// SIMATIC STEP 7 (V5.x) project EMPTYING
// program: S7 Program(1)

SYMBOL_TABLE
"EMPTYING_CYCLE"	FB 148	FB 148	// Цикл опустошения илоуплотнителей
END_SYMBOL_TABLE

FUNCTION_BLOCK "EMPTYING_CYCLE"	// FB 148
TITLE = Блок управления циклами слива
//Используемая переферия:
//Таймеры:
//Счетчики:
//
//
////Авария по сливу, насосы откачки не запустились
////Фильтр аварий в режимах работы чтобы запустить слив на одном затворе
AUTHOR : ETSystem
VERSION : 0.1
VAR_INPUT
  G32_OPENED : BOOL ;	//Затвор 3-2 открыт
  G32_CLOSED : BOOL ;	//Затвор 3-2 закрыт
  G32_FAULT : BOOL ;	//Авария затвора 3-2
  G34_OPENED : BOOL ;	//Затвор 3-4 открыт
  G34_CLOSED : BOOL ;	//Затвор 3-4 закрыт
  G34_FAULT : BOOL ;	//Авария затвора 3-4
  WT_ONOFF : BOOL ;	//Цикл ожидания активен/нет
  AUTO_ONOFF : BOOL ;	//Автоматический режим включен
  LEVEL_1 : BOOL ;	//Датчик уровня 1 (минимальный уровень)
  LEVEL_2 : BOOL ;	//Датчик уровня 2 (средний уровень)
  LEVEL_3 : BOOL ;	//Датчик уровня 3 (высокий уровень)
  LEVEL_4 : BOOL ;	//Датчик уровня 4 (критический уровень)
  STOP : BOOL ;	//Цикл остановлен
  START : BOOL ;	//Цикл запущен
  EMPTYING_DELAY : INT  := 10;	//Задержка начала слива (в формате TIME)
  G32_CNT_TASK : INT  := 1;	//Количество циклов опорожения затвора 3-2 (0 - 4)
  G34_CNT_TASK : INT  := 1;	//Количество циклов опорожения затвора 3-4 (0 - 4)
END_VAR
VAR_OUTPUT
  QG32_OPENING : BOOL ;	//Команда на открытие затвора 3-2
  QG32_CLOSING : BOOL ;	//Команда на закрытие затвора 3-2
  QG32_FAULT : BOOL ;	//Авария на затворе 3-2
  QG34_OPENING : BOOL ;	//Команда на открытие затвора 3-4
  QG34_CLOSING : BOOL ;	//Команда на закрытие затвора 3-4
  QG34_FAULT : BOOL ;	//Авария на затворе 3-4
  QCOMMON_FAULT : BOOL ;	//Общая авария на блоке
  QINIT_OK : BOOL ;	//Работа цикла слива в автоматическом режиме инициализирована
  QG32_ACK : BOOL ;	//Идет слив с затвора 3-2
  QG34_ACK : BOOL ;	//Идет слив с затвора 3-4
  QEMPTYING_ACK : BOOL ;	//Режим слива активен
  QWORK_TIME : INT ;	//Общее время работы слива
END_VAR
VAR_IN_OUT
  G32_CNT : INT ;	//Счетчик циклов слива (затвор 3-2)
  G34_CNT : INT ;	//Счетчик циклов слива (затвор 3-4)
END_VAR
VAR
  LEVEL_FAULT : BOOL ;	//Неисправность датчика уровня
  GATE_FAULT : BOOL ;	//Неисправность одного из затворов (3-2 или 3-4)
  COMMON_FAULT : BOOL ;	//Общая ошибка
  DELAY_OK : BOOL ;	//Задержка цикла слива отработана
  G32_INWORK : BOOL ;	//Затвор 3-2 в работе
  G34_INWORK : BOOL ;	//Затвор 3-4 в работе
  G32_CNT_FLAG : BOOL ;	//Флаг для подсчета циклов слива (затвор 3-2)
  G34_CNT_FLAG : BOOL ;	//Флаг для подсчета циклов слива (затвор 3-4)
  BOTH_FLAG : BOOL ;	//Оба затвора в работе
  INIT_OK : BOOL ;	//Режим слива инициализирован
  MODE : INT ;	//0 - оба неактивны, 1 - оба активны, 2 - активен 3-2, 3 - активен 3-4
  S5T_EMPDELAY : S5TIME ;	//Задержка начала слива (в формате S5T)
  T_EMPDELAY : TIME ;	//Задержка начала слива (в формате TIME)
END_VAR
BEGIN
NETWORK
TITLE = Инициализация цикла (начало)
//Инициализация цикла необходима только один раз при запуске автоматического 
//режима, если инициализация проходит без ошибок, выставляется флаг INIT_OK и на 
//следующем цикле ПЛК готов к автоматическому сливу из илоуплотнителей
//Мы не в автоматическом режиме, уходим сбросив инициализацию цикла если он была
      AN    #AUTO_ONOFF;
//Сбросим признаки аварии после того как выбило в ручной режим
      R     #COMMON_FAULT;
      R     #QCOMMON_FAULT;
      JC    MAN;
//Сбросим сигналы открытия/закрытия если требуется: 
//Сброс сигналов открытия/закрытия  32
      A     #QG32_OPENING;
      A     #G32_OPENED;
      O(;
      A     #QG32_OPENING;
      AN    #G32_OPENED;
      AN    #G32_CLOSED;
      );
      R     #QG32_OPENING;
      A     #QG32_CLOSING;
      A     #G32_CLOSED;
      O(;
      A     #QG32_CLOSING;
      AN    #G32_OPENED;
      AN    #G32_CLOSED;
      );
      R     #QG32_CLOSING;
//Сброс сигналов открытия/закрытия 34
      A     #QG34_OPENING;
      A     #G34_OPENED;
      O(;
      A     #QG34_OPENING;
      AN    #G34_OPENED;
      AN    #G34_CLOSED;
      );
      R     #QG34_OPENING;
      A     #QG34_CLOSING;
      A     #G34_CLOSED;
      O(;
      A     #QG34_CLOSING;
      AN    #G34_OPENED;
      AN    #G34_CLOSED;
      );
      R     #QG34_CLOSING;
//Определяем состояние автоматического режима
      A     #START;
      AN    #INIT_OK;
      JC    INIT;
      AN    #START;
      JC    STOP;
      A     #INIT_OK;
      JC    AUTO;
      JU    N1;
NETWORK
TITLE =  Инициализация цикла (продолжение)
//Выбор верной конфигурации затворов слива:
//Определяем конфигурацию системы слива (единожды). Возможные варианты:
// 1. Активны оба затвора (G32_CNT и G34_CNT) - число их циклов слива не равно 0 
//(MODE 0), выставляется флаг BOTH_FLAG.
// 2. Активен один из затворов (G32_CNT ИЛИ G34_CNT) - число его циклов слива 
//равно 0 (MODE 1, MODE 2).
// 3. Слив запрещен (MODE 0).
// 4. Запись значения в MODE выводится для более удобного наблюдения за тем какой 
//режим был проинициализирован. (для отладки) 
//
//Смена конфигурации режима работы сливов во время исполнения автоматического 
//режима не предусмотрена, и будет инициализирована авария. (Так же она должна 
//быть заблокирована в СКАДА).
//Инициализация (сброс) флагов
INIT: NOP   0;
      L     0;
      T     #G32_CNT;
      T     #G34_CNT;
      SET;
      R     #G32_CNT_FLAG;
      R     #G34_CNT_FLAG;
      R     #G32_INWORK;
      R     #G34_INWORK;
//Сбросим признаки аварии при инициализации
      R     #COMMON_FAULT;
      R     #QCOMMON_FAULT;
//Закроем затворы если открыты:
      AN    #G32_CLOSED;
      S     #QG32_CLOSING;
      AN    #G34_CLOSED;
      S     #QG34_CLOSING;
//Оба затвора могут быть в работе (MODE 1)
      AN    #G32_FAULT;
      AN    #G34_FAULT;
      A(;
      L     #G32_CNT_TASK;
      L     0;
      <>I;
      );
      A(;
      L     #G34_CNT_TASK;
      L     0;
      <>I;
      );
      L     1;
//Инициализаруем активный затвор и флаг того что
//в работе оба затвора
      S     #G32_INWORK;
      S     #BOTH_FLAG;
      JC    MSEL;
//Затвор 3-2 может быть в работе (MODE 2)
      AN    #G32_FAULT;
      A(;
      L     #G32_CNT_TASK;
      L     0;
      <>I;
      );
      L     2;
      S     #G32_INWORK;
      R     #BOTH_FLAG;
      JC    MSEL;
//Затвор 3-4 может быть в работе (MODE 3)
      AN    #G34_FAULT;
      A(;
      L     #G34_CNT_TASK;
      L     0;
      <>I;
      );
      L     3;
      S     #G34_INWORK;
      R     #BOTH_FLAG;
      JC    MSEL;
//Ни один из затворов в работе быть не может (MODE 0)
      L     0;
//Задание активной конфигурации
MSEL: T     #MODE;
//Если режим MODE = 0, пропускаем цикл опустошения:
      L     #MODE;
      L     0;
      ==I;
      JC    MOD0;
NETWORK
TITLE =  Инициализация цикла (продолжение)
//Конвертация времени ожидания перед сливом из INT (SCADA) в S5T (Siemens) с 
//помощью функции FC40, через переменную типа TIME (IEC). Итого вое время в 
//секундах. Задание из SCADA в секундах.
      L     #EMPTYING_DELAY;
      ITD;
      L     L#1000;
      *D;
      T     #T_EMPDELAY;
      CALL  FC 40 (
           $1                       := #T_EMPDELAY,
           $2                       := #S5T_EMPDELAY);
NETWORK
TITLE = Инициализация цикла слива (конец)
//Если включен автоматический режим, и бак пуст (не один из датчиков не включен)
      A     #AUTO_ONOFF;
      A     #G32_CLOSED;
      A     #G34_CLOSED;
      AN    #LEVEL_1;
      AN    #LEVEL_2;
      AN    #LEVEL_3;
      AN    #LEVEL_4;
      S     #INIT_OK;
      JCN   N1;
NETWORK
TITLE = Автоматический режим слива илоуплотнителей (начало)
//Сброс сигналов на открытие или закрытие затворов
AUTO: NOP   0;
NETWORK
TITLE = Переинициализация автомата
//Если мы не в режиме ожидания, сбросим таймер и флаг окончания задержки, а так 
//же обнулим счетчики сливов по каждому из затворов.
      AN    #WT_ONOFF;
      R     T 5;
      R     #DELAY_OK;
      JCN   NX1;
//Обнуление счетчиков
      L     0;
      T     #G32_CNT;
      T     #G34_CNT;
//Сброс флагов
      SET;
      R     #G32_CNT_FLAG;
      R     #G34_CNT_FLAG;
//Переинициализация активного затвора
      A     #BOTH_FLAG;
      O(;
      L     #MODE;
      L     2;
      ==I;
      );
      S     #G32_INWORK;
      L     #MODE;
      L     3;
      ==I;
      S     #G34_INWORK;
NETWORK
TITLE = Определение аварий
//Определяем текущие аварии, при их возникновении цикл налива-слива должен быть 
//остановлен, для этого необходимо использовать блок налива (FB_xxx) как блок 
//общей задачи автоматического режима. Вопрос с ручным - автоматическим режимом 
//на затворах 3-2 и 3-4 требует отдельного рассмотрения. 
//
//Подумать над общей неисправностью.
NX1:  NOP   0;
//Проверяем верно ли работает линейка датчиков 
//Неисправность датчика первого уровня:
//(НЕ Уровень1 И (Уровень2 ИЛИ Уровень3 ИЛИ Уровень4))
      AN    #LEVEL_1;
      A(;
      O     #LEVEL_2;
      O     #LEVEL_3;
      O     #LEVEL_4;
      );
      O;
//Или их непоследовательное включение:
//(Уровень1 И ((Уровень3 И НЕ Уровень2) ИЛИ (Уровень4 И НЕ Уровень3))
      A     #LEVEL_1;
      A(;
      A     #LEVEL_3;
      AN    #LEVEL_2;
      O;
      A     #LEVEL_4;
      AN    #LEVEL_3;
      );
      =     #LEVEL_FAULT;
//Проверяем наличие аварий на затворах 3-2 и 3-4:
//Неисправности затворов:
//     O     #G32_FAULT
//      O     #G34_FAULT
//      =     #GATE_FAULT
//Выдаем аварии по затвору в зависимости от режима работы:
//Режим 1:
      L     #MODE;
      L     1;
      ==I;
      JC    ERR1;
//Режим 2:
      L     #MODE;
      L     2;
      ==I;
      JC    ERR2;
//Режим 3:
      L     #MODE;
      L     3;
      ==I;
      JC    ERR3;
//Нет аварий по затворам
      JU    ERRC;
ERR1: NOP   0;
      O     #G32_FAULT;
      O     #G34_FAULT;
      =     #GATE_FAULT;
      JU    ERRC;
ERR2: NOP   0;
      A     #G32_FAULT;
      =     #GATE_FAULT;
      JU    ERRC;
ERR3: NOP   0;
      A     #G34_FAULT;
      =     #GATE_FAULT;
ERRC: NOP   0;
//Общая неисправность:
      O     #LEVEL_FAULT;
      O     #GATE_FAULT;
      =     #COMMON_FAULT;
      JC    ALRM;
NETWORK
TITLE = Задержка начала первого цикла слива
//Если активировался режим ожидания налива (WT_ONOFF = 1) И с определенной 
//конфигурацией (MODE != 0) -  дополнительная проверка, которую можно убрать.
//То запускаем таймер задержки слива (T5 - 
//DELAY_EMPTYING), S_ODT - считает пока на его входе 1, если она пропадает, счет 
//останавливается и при восcтановлении сигнала запускается заново. 
      A     #DELAY_OK;
      JC    NX2;
      A     #WT_ONOFF;
      A(;
      L     #MODE;
      L     0;
      <>I;
      );
      L     #S5T_EMPDELAY;
      SD    T 5;
      A     T 5;
      S     #DELAY_OK;
      S     #QEMPTYING_ACK;
NETWORK
TITLE = Цикл слива с обоих затворов
//В зависимости от режима работы возможно нескольк сценариев слива:
// 1. Через оба клапана, сначала n циклов с 3-2, затем n циклов с 3-4
// 2. n циклов через один клапан (3-2 или 3-4) 
NX2:  NOP   0;
//Если задержка после заполнения не отработала, то начинать процесс слива
//нельзя, ожидаем поднятие флага DELAY_OK
      AN    #DELAY_OK;
      JC    N1;
//Если G32 в работе, инициализируем слив
      A     #G32_INWORK;
      AN    #G32_CNT_FLAG;
      JC    G32E;
//Цикл отработал и затвор закрылся
      A     #G32_CNT_FLAG;
      A     #G32_CLOSED;
      JC    G32C;
//Если G34 в работе, инициализируем слив
      A     #G34_INWORK;
      AN    #G34_CNT_FLAG;
      JC    G34E;
//Цикл отработал и затвор закрылся
      A     #G34_CNT_FLAG;
      A     #G34_CLOSED;
      JC    G34C;
      JU    N1;
//////////////////////Затвор 3-2/////////////////////
//Открытие и закрытие затвора
G32E: NOP   0;
//Открываем затвор если уровень в баке опустился до нужного уровня
//И затвор открыт
      AN    #LEVEL_1;
      A     #G32_CLOSED;
      S     #QG32_OPENING;
      S     #QG32_ACK;
//Закрываем затвор если уровень в баке поднялся до нужного уровня
//И затвор открыт, так же устанавливаем флаг для подсчета циклов
      A     #LEVEL_2;
      A     #G32_OPENED;
      S     #QG32_CLOSING;
      S     #G32_CNT_FLAG;
      JU    N1;
//Подсчет циклов и условие выхода (смены затвора)
G32C: NOP   0;
//Номер прошедшего цикла слива определяется по факту закрытия затвора
//так же определяется прошло ли нужное количество сливов и переключается
//активный затвор (если требуется), флаг счетчика сливов сбрасывается
      R     #G32_CNT_FLAG;
      L     1;
      L     #G32_CNT;
      +I;
      T     #G32_CNT;
//Был выполнен последний цикл слива на текущем затворе
      L     #G32_CNT;
      L     #G32_CNT_TASK;
      ==I;
      R     #G32_INWORK;
      R     #QG32_ACK;
//Если требуется слив с обоих затворов, инициализируем 3-4 
      A     #BOTH_FLAG;
      S     #G34_INWORK;
      AN    #BOTH_FLAG;
      R     #QEMPTYING_ACK;
//Иначе заканчиваев цикл сливов в текущем периоде ожидания
      JU    N1;
//////////////////////Затвор 3-4/////////////////////
//Открытие и закрытие затвора
G34E: NOP   0;
//Открываем затвор
      AN    #LEVEL_1;
      A     #G34_CLOSED;
      S     #QG34_OPENING;
      S     #QG34_ACK;
//Закрываем затвор
      A     #LEVEL_2;
      A     #G34_OPENED;
      S     #QG34_CLOSING;
      S     #G34_CNT_FLAG;
      JU    N1;
//Подсчет циклов и условие выхода (смены затвора)
G34C: NOP   0;
      R     #G34_CNT_FLAG;
      L     1;
      L     #G34_CNT;
      +I;
      T     #G34_CNT;
      L     #G34_CNT;
      L     #G34_CNT_TASK;
      ==I;
      R     #G34_INWORK;
      R     #QG34_ACK;
      R     #QEMPTYING_ACK;
//Заканчиваем цикл сливов в текущем периоде ожидания
      JU    N1;
NETWORK
TITLE = Общий таймер
//Общий таймер активируется в период активности режима слива и считает суммарное 
//время слива за весь период работы цикла слива/налива, в минутах.
NETWORK
TITLE = STOP
STOP: NOP   0;
      R     #INIT_OK;
      R     #QG32_ACK;
      R     #QG34_ACK;
      R     #QEMPTYING_ACK;
//Если нажали кнопку STOP - закрываем затворы
      AN    #G32_CLOSED;
      A     #QG32_CLOSING;
      AN    #G34_CLOSED;
      A     #QG34_CLOSING;
      JC    N1;
NETWORK
TITLE = Обработка выходных параметров блока
ALRM: NOP   0;
//Устанавливаем общий аварийный выход блока 
      A     #COMMON_FAULT;
      =     #QCOMMON_FAULT;
//В качестве диагностики определим аварийный затвор слива
      A     #G32_FAULT;
      =     #QG32_FAULT;
      A     #G34_FAULT;
      =     #QG34_FAULT;
//Сбросим таймер и флаг удачной задержки
      SET;
      R     T 5;
      R     #DELAY_OK;
//Цикл опустошения запрещен, по хорошему это надо идентифицировать
//как аварию и запрещать запуск автоматического режима
MOD0: NOP   0;
NETWORK
TITLE = Переход в ручной режим
MAN:  NOP   0;
      AN    #AUTO_ONOFF;
      R     #INIT_OK;
      R     #QG32_ACK;
      R     #QG34_ACK;
      R     #QEMPTYING_ACK;
      R     #G32_CNT_FLAG;
      R     #G34_CNT_FLAG;
      R     #G32_INWORK;
      R     #G34_INWORK;
//Сбросим сигналы на открытие-закрытие при переходе в ручной режим
      R     #QG32_OPENING;
      R     #QG32_CLOSING;
      R     #QG34_OPENING;
      R     #QG34_CLOSING;
      L     0;
      T     #G32_CNT;
      T     #G34_CNT;
NETWORK
TITLE =
N1:   NOP   0;
END_FUNCTION_BLOCK

ORGANIZATION_BLOCK OB 1
TITLE = "Main Program Sweep (Cycle)"
VERSION : 0.1
VAR_TEMP
  OB1_EV_CLASS : BYTE ;	//Bits 0-3 = 1 (Coming event), Bits 4-7 = 1 (Event class 1)
  OB1_SCAN_1 : BYTE ;	//1 (Cold restart scan 1 of OB 1), 3 (Scan 2-n of OB 1)
  OB1_PRIORITY : BYTE ;	//Priority of OB Execution
  OB1_OB_NUMBR : BYTE ;	//1 (Organization block 1, OB1)
  OB1_RESERVED_1 : BYTE ;	//Reserved for system
  OB1_RESERVED_2 : BYTE ;	//Reserved for system
  OB1_PREV_CYCLE : INT ;	//Cycle time of previous OB1 scan (milliseconds)
  OB1_MIN_CYCLE : INT ;	//Minimum cycle time of OB1 (milliseconds)
  OB1_MAX_CYCLE : INT ;	//Maximum cycle time of OB1 (milliseconds)
  OB1_DATE_TIME : DATE_AND_TIME ;	//Date and time OB1 started
END_VAR
BEGIN
// (block stored without names or comments; labels and parameter names are numbered)
END_ORGANIZATION_BLOCK
